// ---- StateMachine/UnifiedProgram/Transitions/SuspendedToHaltedUnifiedProgramTransition.TcPOU
FUNCTION_BLOCK SuspendedToHaltedUnifiedProgramTransition EXTENDS SuspendedToHaltedProgramTransition
VAR
	{attribute 'OPC.UA.DA' := '0'}
	_ClassName : STRING := __POUNAME();
END_VAR

{attribute 'monitoring' := 'call'}
PROPERTY ClassName : STRING
GET
ClassName := _ClassName;
END_GET
END_PROPERTY

END_FUNCTION_BLOCK

// ---- StateMachine/UnifiedProgram/Transitions/SuspendedToReadyUnifiedProgramTransition.TcPOU
FUNCTION_BLOCK SuspendedToReadyUnifiedProgramTransition EXTENDS SuspendedToReadyProgramTransition
VAR
	{attribute 'OPC.UA.DA' := '0'}
	_ClassName : STRING := __POUNAME();
END_VAR

{attribute 'monitoring' := 'call'}
PROPERTY ClassName : STRING
GET
ClassName := _ClassName;
END_GET
END_PROPERTY

END_FUNCTION_BLOCK

// ---- StateMachine/UnifiedProgram/UnifiedProgramStepExecutor.TcPOU
{attribute 'no_explicit_call' := 'do not call this function block directly'} 
{attribute 'OPC.UA.DA' := '0'}
FUNCTION_BLOCK INTERNAL UnifiedProgramStepExecutor EXTENDS ToolkitObject
VAR
	_ClassName : STRING := __POUNAME();

	_StateMachine : REFERENCE TO UnifiedProgramStateMachine;
	
	_ExecutedSteps : ARRAY [0..UnifiedProgramConstants.MaxStepCount - 1] OF UNIFIED_PROGRAM_EXECUTED_STEP;
	_ExecutedStepCount : INT;
	_ExecutedStep : REFERENCE TO UNIFIED_PROGRAM_EXECUTED_STEP;	
END_VAR

{attribute 'monitoring' := 'call'}
PROPERTY ClassName : STRING
GET
ClassName := _ClassName;
END_GET
END_PROPERTY

METHOD FB_init : BOOL
VAR_INPUT
	bInitRetains : BOOL; // if TRUE, the retain variables are initialized (warm start / cold start)
	bInCopyCode : BOOL; // if TRUE, the instance afterwards gets moved into the copy code (online change)
	stateMachine : REFERENCE TO UnifiedProgramStateMachine;
END_VAR
_StateMachine REF= stateMachine;
END_METHOD

METHOD Reset 
VAR
	i : DINT;
END_VAR
FOR i := 0 TO UnifiedProgramConstants.MaxStepCount - 1 DO
	_ExecutedSteps[i].StepIndex := -1;
	_ExecutedSteps[i].Step REF= 0;
END_FOR

_ExecutedStepCount := 0;
_ExecutedStep REF= 0;
END_METHOD

END_FUNCTION_BLOCK
